PROGRAM LM_State_MC_TCP
VAR
END_VAR

// NETWORK 1

END_PROGRAM

(* stored: Version 1.1.0.1, ProductVersion 3.1.4024.0
   POU LM_State_MC_TCP: Id {b239ecf3-62f6-4772-a148-96f3cfe77a8b}, SpecialFunc None *)
